{attribute 'analysis' := '-33'} // inhibit unused variable warning
FUNCTION_BLOCK TestSuite_AssertTests
VAR
    TestRunner                               : T_TestRunner(TestSuiteName := 'TestSuite_AssertTests', Verbose := FALSE);
    Test_AssertEqualsDetects_INTS_ThatDiffer : Test_AssertEqualsDetects_INTS_ThatDiffer(TestRunner);
    Test_AssertEquals_STRING                 : Test_AssertEquals_STRING(TestRunner);
END_VAR

TestRunner.CyclicUpdate();

END_FUNCTION_BLOCK

(* stored: Version 1.1.0.1, ProductVersion 3.1.4024.12
   POU TestSuite_AssertTests: Id {79ad6bd5-b125-43a8-80f3-d60ad2c36432}, SpecialFunc None *)
